(* Schneider Machine Expert - Basic project Timer 3 BLK, file version 1.7.0.0 *)
(* ProjectInformations: Name=New project *)

HARDWARE
  Cpu 0: TM221M16R/G
  EthernetConfiguration: NetworkName=M221, IpAllocationMode=FixedAddress, IpAddress=0.0.0.0, SubnetMask=0.0.0.0
  SerialLineConfiguration: Baud=Baud19200, Parity=ParityEven, DataBits=DataBits8, StopBits=StopBits1, PhysicalMedium=PhysicalMediumRs485, TransmissionMode=TransmissionModeModbusRtu, SlaveId=1, Addressing=SlaveAddressing
  MastTask: UsePeriodScanMode=false, PeriodScan=100
  FastTask: Period=255
  CpuBehavior: StartingMode=StartAsPreviousState, AutoSaveRamOnEeprom=true, WatchdogPeriod=250

SYMBOLS  (address, symbol, comment, settings)
  %TM0        "T1"  [Preset=1, Base=OneSecond]

POU New POU
  (* SectionNumber=1 *)

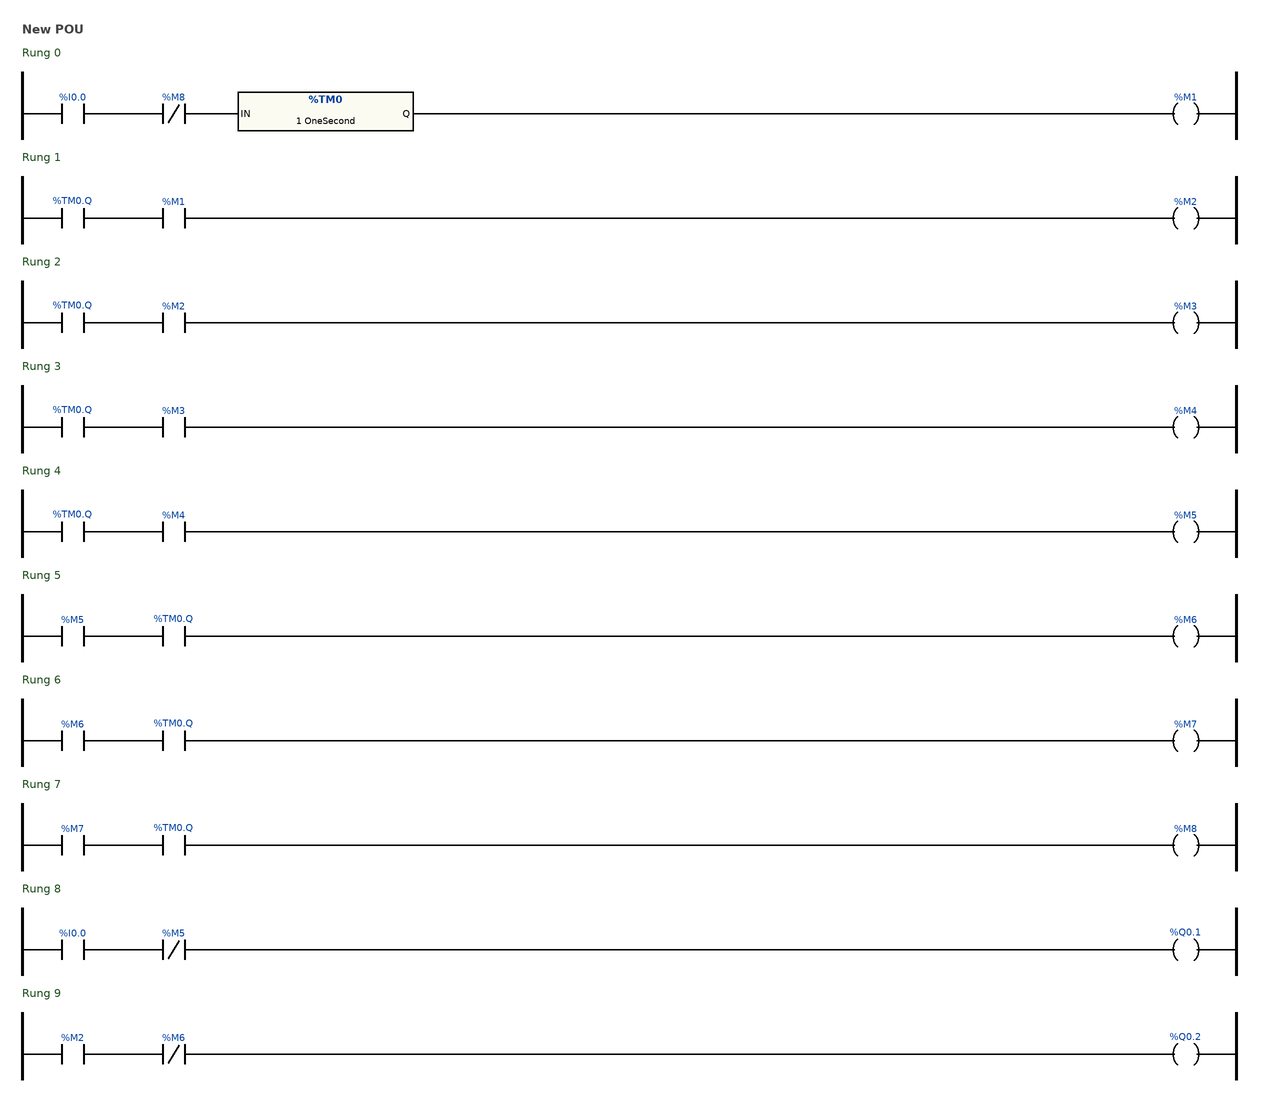

// Rung 0
  BLK %TM0
  LD %I0.0
  ANDN %M8
  IN
  OUT_BLK
  LD Q
  ST %M1
  END_BLK
  // as ST:
  //   %TM0(IN := %I0.0 AND NOT %M8);
  //   %M1 := %TM0.Q;

// Rung 1
  LD %TM0.Q
  AND %M1
  ST %M2
  // as ST:
  //   %M2 := %TM0.Q AND %M1;

// Rung 2
  LD %TM0.Q
  AND %M2
  ST %M3
  // as ST:
  //   %M3 := %TM0.Q AND %M2;

// Rung 3
  LD %TM0.Q
  AND %M3
  ST %M4
  // as ST:
  //   %M4 := %TM0.Q AND %M3;

// Rung 4
  LD %TM0.Q
  AND %M4
  ST %M5
  // as ST:
  //   %M5 := %TM0.Q AND %M4;

// Rung 5
  LD %M5
  AND %TM0.Q
  ST %M6
  // as ST:
  //   %M6 := %M5 AND %TM0.Q;

// Rung 6
  LD %M6
  AND %TM0.Q
  ST %M7
  // as ST:
  //   %M7 := %M6 AND %TM0.Q;

// Rung 7
  LD %M7
  AND %TM0.Q
  ST %M8
  // as ST:
  //   %M8 := %M7 AND %TM0.Q;

// Rung 8
  LD %I0.0
  ANDN %M5
  ST %Q0.1
  // as ST:
  //   %Q0.1 := %I0.0 AND NOT %M5;

// Rung 9
  LD %M2
  ANDN %M6
  ST %Q0.2
  // as ST:
  //   %Q0.2 := %M2 AND NOT %M6;

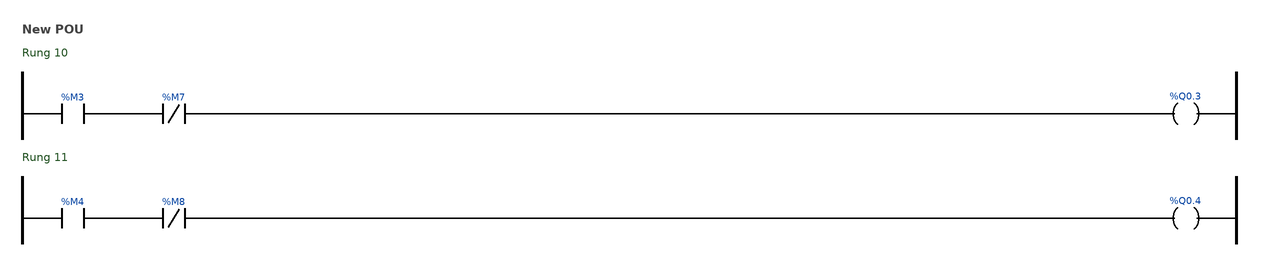

// Rung 10
  LD %M3
  ANDN %M7
  ST %Q0.3
  // as ST:
  //   %Q0.3 := %M3 AND NOT %M7;

// Rung 11
  LD %M4
  ANDN %M8
  ST %Q0.4
  // as ST:
  //   %Q0.4 := %M4 AND NOT %M8;
